FUNCTION_BLOCK Section1Ctrl (* Basic Function Block Type *)
  (* Standard: 61499-2 *)
  (* Version 0.0, 5/27/2018, MIA, nxtControl GmbH, Template *)
  PACKAGE Main;
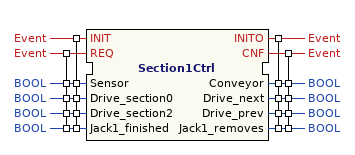
  EVENT_INPUT
    INIT WITH Sensor, Drive_section0, Drive_section2, Jack1_finished; (* Initialization Request *)
    REQ WITH Sensor, Drive_section0, Drive_section2, Jack1_finished; (* Normal Execution Request *)
  END_EVENT
  EVENT_OUTPUT
    INITO WITH Conveyor, Drive_next, Drive_prev, Jack1_removes; (* Initialization Confirm *)
    CNF WITH Conveyor, Drive_next, Drive_prev, Jack1_removes; (* Execution Confirmation *)
  END_EVENT
  VAR_INPUT
    Sensor : BOOL; (* Input event qualifier *)
    Drive_section0 : BOOL;
    Drive_section2 : BOOL;
    Jack1_finished : BOOL;
  END_VAR
  VAR_OUTPUT
    Conveyor : BOOL; (* Output event qualifier *)
    Drive_next : BOOL;
    Drive_prev : BOOL;
    Jack1_removes : BOOL;
  END_VAR
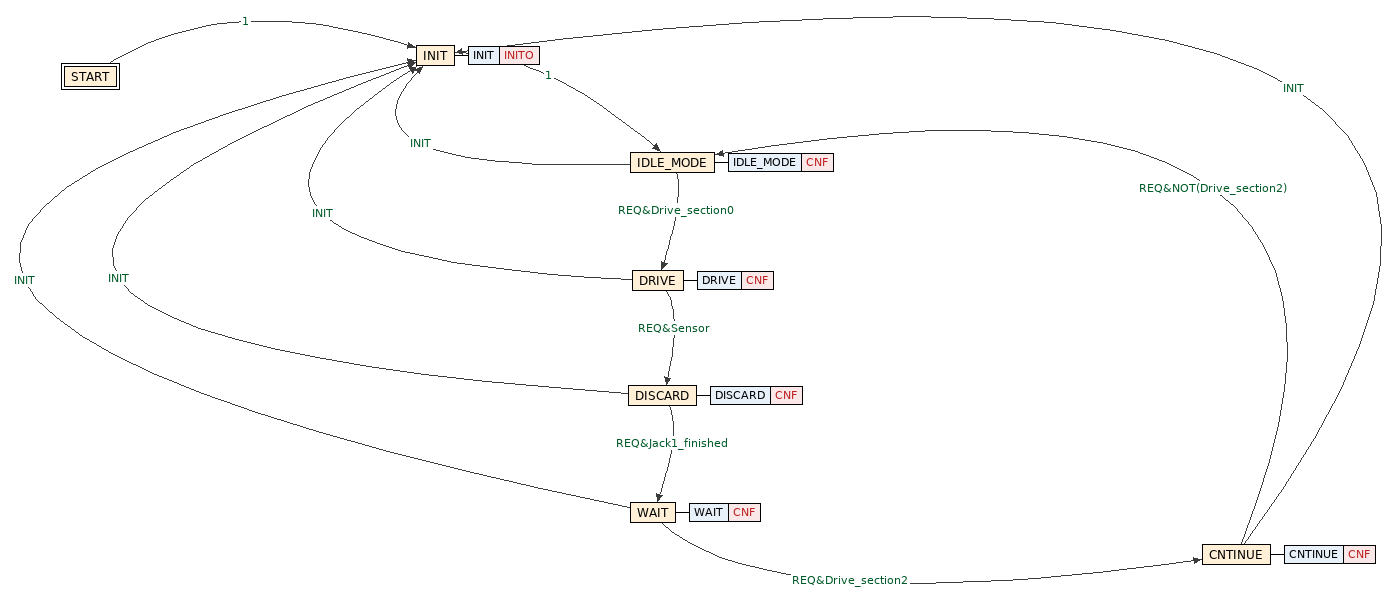
  EC_STATES
    START; (* Initial State *)
    INIT : INIT -> INITO; (* Initialization *)
    IDLE_MODE : IDLE_MODE -> CNF;
    DRIVE : DRIVE -> CNF;
    DISCARD : DISCARD -> CNF;
    WAIT : WAIT -> CNF;
    CNTINUE : CNTINUE -> CNF;
  END_STATES
  EC_TRANSITIONS
    START TO INIT := 1;
    INIT TO IDLE_MODE := 1;
    IDLE_MODE TO INIT := INIT;
    IDLE_MODE TO DRIVE := REQ&Drive_section0;
    DRIVE TO INIT := INIT;
    DRIVE TO DISCARD := REQ&Sensor;
    DISCARD TO INIT := INIT;
    DISCARD TO WAIT := REQ&Jack1_finished;
    WAIT TO INIT := INIT;
    WAIT TO CNTINUE := REQ&Drive_section2;
    CNTINUE TO IDLE_MODE := REQ&NOT(Drive_section2);
    CNTINUE TO INIT := INIT;
  END_TRANSITIONS
  ALGORITHM INIT IN ST: (* Initialization algorithm *)
;
Conveyor := FALSE;
Jack1_removes := FALSE;
Drive_prev := FALSE;
Drive_next := FALSE;
  END_ALGORITHM
  ALGORITHM IDLE_MODE IN ST:
;
Conveyor := FALSE;
Jack1_removes := FALSE;
Drive_prev := TRUE;
Drive_next := FALSE;
  END_ALGORITHM
  ALGORITHM DRIVE IN ST:
;
Conveyor := TRUE;
Jack1_removes := FALSE;
Drive_prev := TRUE;
Drive_next := FALSE;
  END_ALGORITHM
  ALGORITHM DISCARD IN ST:
;
Conveyor := FALSE;
Jack1_removes := TRUE;
Drive_prev := FALSE;
Drive_next := FALSE;
  END_ALGORITHM
  ALGORITHM WAIT IN ST:
;
Conveyor := FALSE;
Jack1_removes := FALSE;
Drive_prev := FALSE;
Drive_next := TRUE;
  END_ALGORITHM
  ALGORITHM CNTINUE IN ST:
;
Conveyor := TRUE;
Jack1_removes := FALSE;
Drive_prev := TRUE;
Drive_next := TRUE;
  END_ALGORITHM
END_FUNCTION_BLOCK
